FUNCTION_BLOCK FB_HE_SATT_FilterHolderSelectorTestDouble IMPLEMENTS I_HE_SATT_FilterHolderSelector
VAR
    abSelectedHolder : ARRAY[1..PL_HE_SATT_Parameters.nNumHolders] OF BOOL;
END_VAR


METHOD DeselectHolder
VAR_INPUT
	nHolderNumber	: INT;
END_VAR

THIS^.abSelectedHolder[nHolderNumber] := FALSE;
END_METHOD


METHOD IsSelected : BOOL
VAR_INPUT
	nHolderNumber	: INT;
END_VAR

IsSelected := THIS^.abSelectedHolder[nHolderNumber];
END_METHOD


METHOD SelectHolder
VAR_INPUT
	nHolderNumber	: INT;
END_VAR

THIS^.abSelectedHolder[nHolderNumber] := TRUE;
END_METHOD

END_FUNCTION_BLOCK

(* stored: Version 1.1.0.1
   POU FB_HE_SATT_FilterHolderSelectorTestDouble: Id {62fc66af-1dd0-41c9-b277-7ece72acbf00}, SpecialFunc None
   Method DeselectHolder: Id {171b5c60-aec1-40cd-b9a6-5433eef26b2a}
   Method IsSelected: Id {f3405b0e-228d-440b-b29e-fa5167707509}
   Method SelectHolder: Id {a98d1e51-3f4d-40d6-ba80-dfbe1e56d8ca} *)
